// TIA Portal V20 export
TYPE "typeCmControlNodeInterlock"
// stored: Namespace Unit1.Em4
   STRUCT
      sideTapeFixStageAxisX : "LER_typeAxisInterlock";
      sideTapeFixStageAxisC : "LER_typeAxisInterlock";
      sideTapeAttachmentAxisX : "LER_typeAxisInterlock";
      sideTapeAttachmentAxisY : "LER_typeAxisInterlock";
      sideTapeLoading : "LER_typeTwoWayActuatorInterlock";
      sideTapeLoadingClamp : "LER_typeTwoWayActuatorInterlock";
      sideTapeCutter : "LER_typeTwoWayActuatorInterlock";
      sideTapeCutterClamp : "LER_typeTwoWayActuatorInterlock";
      sideTapeTension : "LER_typeTwoWayActuatorInterlock";
      sideTapeAttachmentLeft : "LER_typeTwoWayActuatorInterlock";
      sideTapeAttachmentRight : "LER_typeTwoWayActuatorInterlock";
      sideTapeAttachmentBtm : "LER_typeTwoWayActuatorInterlock";
      sideTapeFixStage : "LER_typeTwoWayActuatorInterlock";
      sideTapeAttachmentLeftTopVaccum : "LER_typeTwoWayActuatorInterlock";
      sideTapeAttachmentLeftBtmVaccum : "LER_typeTwoWayActuatorInterlock";
      sideTapeAttachmentRightTopVaccum : "LER_typeTwoWayActuatorInterlock";
      sideTapeAttachmentRightBtmVaccum : "LER_typeTwoWayActuatorInterlock";
   END_STRUCT;
END_TYPE
